DATA_BLOCK "ST10_Flow12_A2TableUnloading_iDB"
{ S7_Optimized_Access := 'TRUE' }
VERSION : 0.1
NON_RETAIN
// ATTRIBUTES
// AUTO_NUMBER = False
// BLOCK_NUMBER = 1082
// END_ATTRIBUTES
"ST10_Flow12_A2TableUnloading"

BEGIN

END_DATA_BLOCK

